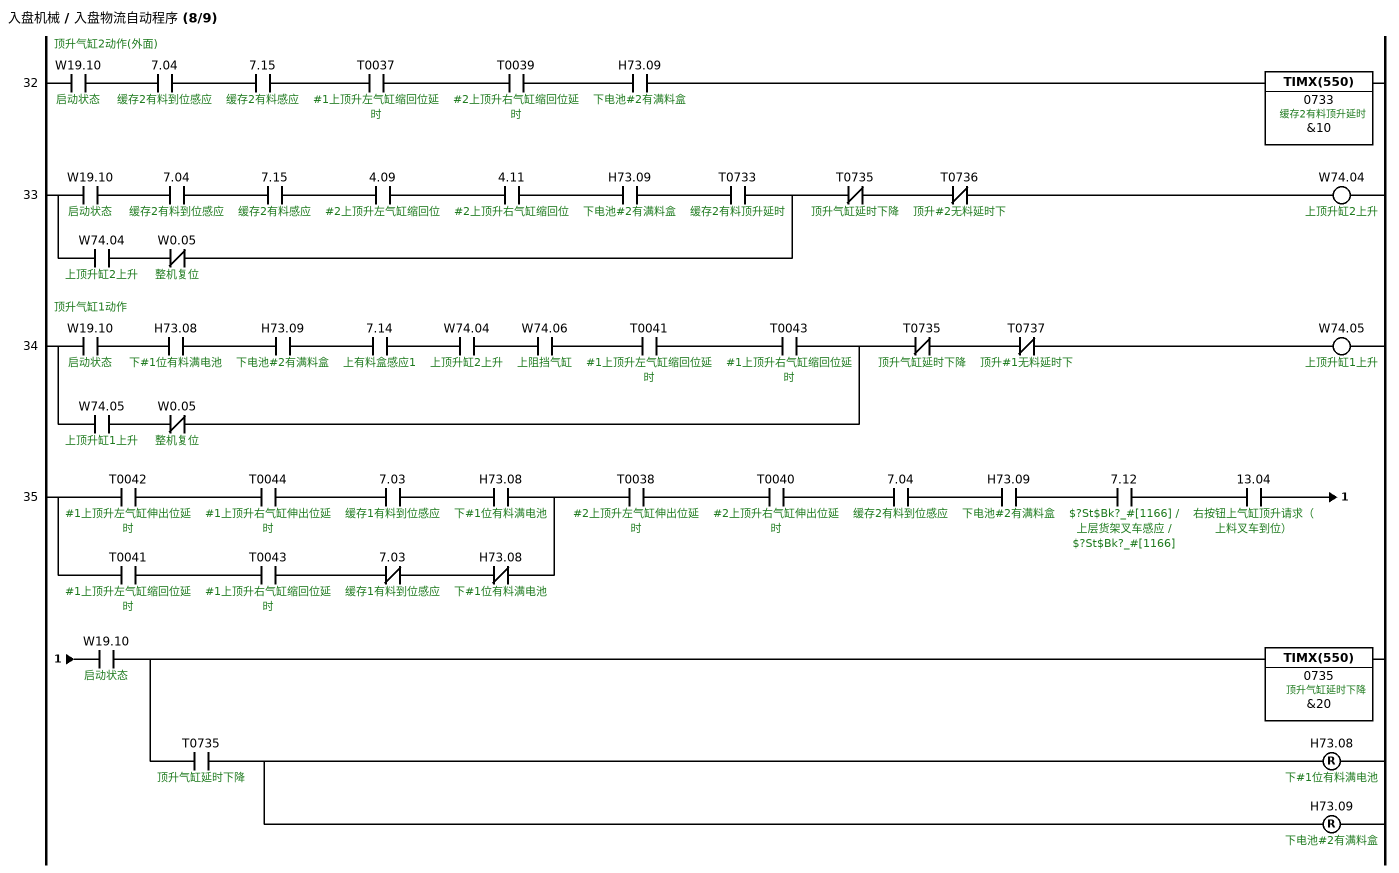
; [picture p240: 入盘机械 / 入盘物流自动程序, rungs 32-35]
; rung 32: 顶升气缸2动作(外面)
LD W19.10  ; 启动状态
AND 7.04  ; 缓存2有料到位感应
AND 7.15  ; 缓存2有料感应
AND T0037  ; #1上顶升左气缸缩回位延时
AND T0039  ; #2上顶升右气缸缩回位延时
AND H73.09  ; 下电池#2有满料盒
TIMX(550) 0733 &10  ; 缓存2有料顶升延时
; rung 33
LD W19.10  ; 启动状态
AND 7.04  ; 缓存2有料到位感应
AND 7.15  ; 缓存2有料感应
AND 4.09  ; #2上顶升左气缸缩回位
AND 4.11  ; #2上顶升右气缸缩回位
AND H73.09  ; 下电池#2有满料盒
AND T0733  ; 缓存2有料顶升延时
LD W74.04  ; 上顶升缸2上升
ANDNOT W0.05  ; 整机复位
ORLD
ANDNOT T0735  ; 顶升气缸延时下降
ANDNOT T0736  ; 顶升#2无料延时下
OUT W74.04  ; 上顶升缸2上升
; rung 34: 顶升气缸1动作
LD W19.10  ; 启动状态
AND H73.08  ; 下#1位有料满电池
AND H73.09  ; 下电池#2有满料盒
AND 7.14  ; 上有料盒感应1
AND W74.04  ; 上顶升缸2上升
AND W74.06  ; 上阻挡气缸
AND T0041  ; #1上顶升左气缸缩回位延时
AND T0043  ; #1上顶升右气缸缩回位延时
LD W74.05  ; 上顶升缸1上升
ANDNOT W0.05  ; 整机复位
ORLD
ANDNOT T0735  ; 顶升气缸延时下降
ANDNOT T0737  ; 顶升#1无料延时下
OUT W74.05  ; 上顶升缸1上升
; rung 35
LD T0042  ; #1上顶升左气缸伸出位延时
AND T0044  ; #1上顶升右气缸伸出位延时
AND 7.03  ; 缓存1有料到位感应
AND H73.08  ; 下#1位有料满电池
LD T0041  ; #1上顶升左气缸缩回位延时
AND T0043  ; #1上顶升右气缸缩回位延时
ANDNOT 7.03  ; 缓存1有料到位感应
ANDNOT H73.08  ; 下#1位有料满电池
ORLD
AND T0038  ; #2上顶升左气缸伸出位延时
AND T0040  ; #2上顶升右气缸伸出位延时
AND 7.04  ; 缓存2有料到位感应
AND H73.09  ; 下电池#2有满料盒
AND 7.12  ; $?St$Bk?_#[1166] / 上层货架叉车感应 / $?St$Bk?_#[1166]
AND 13.04  ; 右按钮上气缸顶升请求（上料叉车到位）
AND W19.10  ; 启动状态
TIMX(550) 0735 &20  ; 顶升气缸延时下降
AND T0735  ; 顶升气缸延时下降
RSET H73.08  ; 下#1位有料满电池
RSET H73.09  ; 下电池#2有满料盒

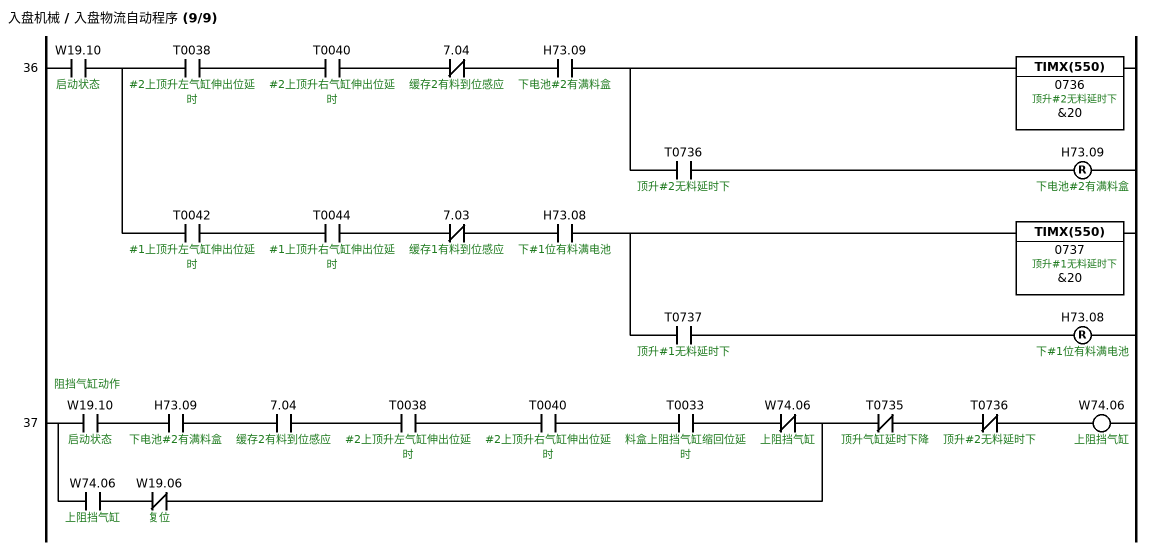
; rung 36
LD W19.10  ; 启动状态
OUT TR0
AND T0038  ; #2上顶升左气缸伸出位延时
AND T0040  ; #2上顶升右气缸伸出位延时
ANDNOT 7.04  ; 缓存2有料到位感应
AND H73.09  ; 下电池#2有满料盒
TIMX(550) 0736 &20  ; 顶升#2无料延时下
AND T0736  ; 顶升#2无料延时下
RSET H73.09  ; 下电池#2有满料盒
LD TR0
AND T0042  ; #1上顶升左气缸伸出位延时
AND T0044  ; #1上顶升右气缸伸出位延时
ANDNOT 7.03  ; 缓存1有料到位感应
AND H73.08  ; 下#1位有料满电池
TIMX(550) 0737 &20  ; 顶升#1无料延时下
AND T0737  ; 顶升#1无料延时下
RSET H73.08  ; 下#1位有料满电池
; rung 37: 阻挡气缸动作
LD W19.10  ; 启动状态
AND H73.09  ; 下电池#2有满料盒
AND 7.04  ; 缓存2有料到位感应
AND T0038  ; #2上顶升左气缸伸出位延时
AND T0040  ; #2上顶升右气缸伸出位延时
AND T0033  ; 料盒上阻挡气缸缩回位延时
ANDNOT W74.06  ; 上阻挡气缸
LD W74.06  ; 上阻挡气缸
ANDNOT W19.06  ; 复位
ORLD
ANDNOT T0735  ; 顶升气缸延时下降
ANDNOT T0736  ; 顶升#2无料延时下
OUT W74.06  ; 上阻挡气缸

### Section 伺服参数设定

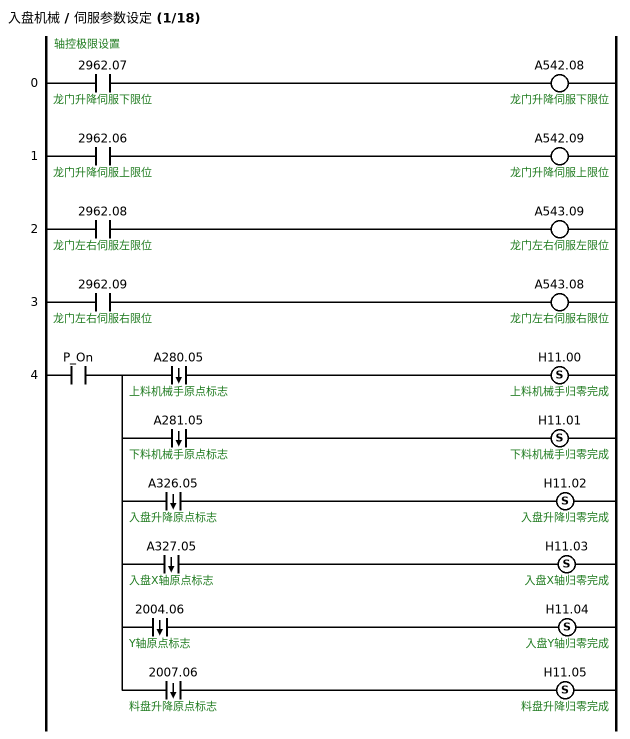
; rung 0: 轴控极限设置
LD 2962.07  ; 龙门升降伺服下限位
OUT A542.08  ; 龙门升降伺服下限位
; rung 1
LD 2962.06  ; 龙门升降伺服上限位
OUT A542.09  ; 龙门升降伺服上限位
; rung 2
LD 2962.08  ; 龙门左右伺服左限位
OUT A543.09  ; 龙门左右伺服左限位
; rung 3
LD 2962.09  ; 龙门左右伺服右限位
OUT A543.08  ; 龙门左右伺服右限位
; rung 4
LD P_On
OUT TR0
%AND A280.05  ; 上料机械手原点标志
SET H11.00  ; 上料机械手归零完成
LD TR0
%AND A281.05  ; 下料机械手原点标志
SET H11.01  ; 下料机械手归零完成
LD TR0
%AND A326.05  ; 入盘升降原点标志
SET H11.02  ; 入盘升降归零完成
LD TR0
%AND A327.05  ; 入盘X轴原点标志
SET H11.03  ; 入盘X轴归零完成
LD TR0
%AND 2004.06  ; Y轴原点标志
SET H11.04  ; 入盘Y轴归零完成
LD TR0
%AND 2007.06  ; 料盘升降原点标志
SET H11.05  ; 料盘升降归零完成

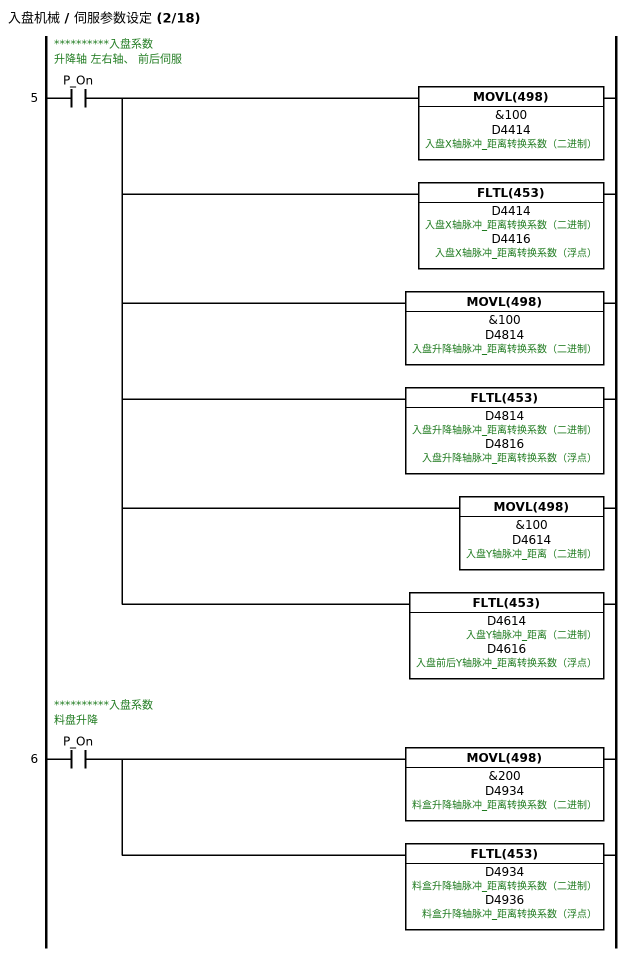
; rung 5: **********入盘系数 / 升降轴 左右轴、 前后伺服
LD P_On
MOVL(498) &100 D4414  ; 入盘X轴脉冲_距离转换系数（二进制）
FLTL(453) D4414 D4416  ; 入盘X轴脉冲_距离转换系数（二进制）, 入盘X轴脉冲_距离转换系数（浮点）
MOVL(498) &100 D4814  ; 入盘升降轴脉冲_距离转换系数（二进制）
FLTL(453) D4814 D4816  ; 入盘升降轴脉冲_距离转换系数（二进制）, 入盘升降轴脉冲_距离转换系数（浮点）
MOVL(498) &100 D4614  ; 入盘Y轴脉冲_距离（二进制）
FLTL(453) D4614 D4616  ; 入盘Y轴脉冲_距离（二进制）, 入盘前后Y轴脉冲_距离转换系数（浮点）
; rung 6: **********入盘系数 / 料盘升降
LD P_On
MOVL(498) &200 D4934  ; 料盒升降轴脉冲_距离转换系数（二进制）
FLTL(453) D4934 D4936  ; 料盒升降轴脉冲_距离转换系数（二进制）, 料盒升降轴脉冲_距离转换系数（浮点）

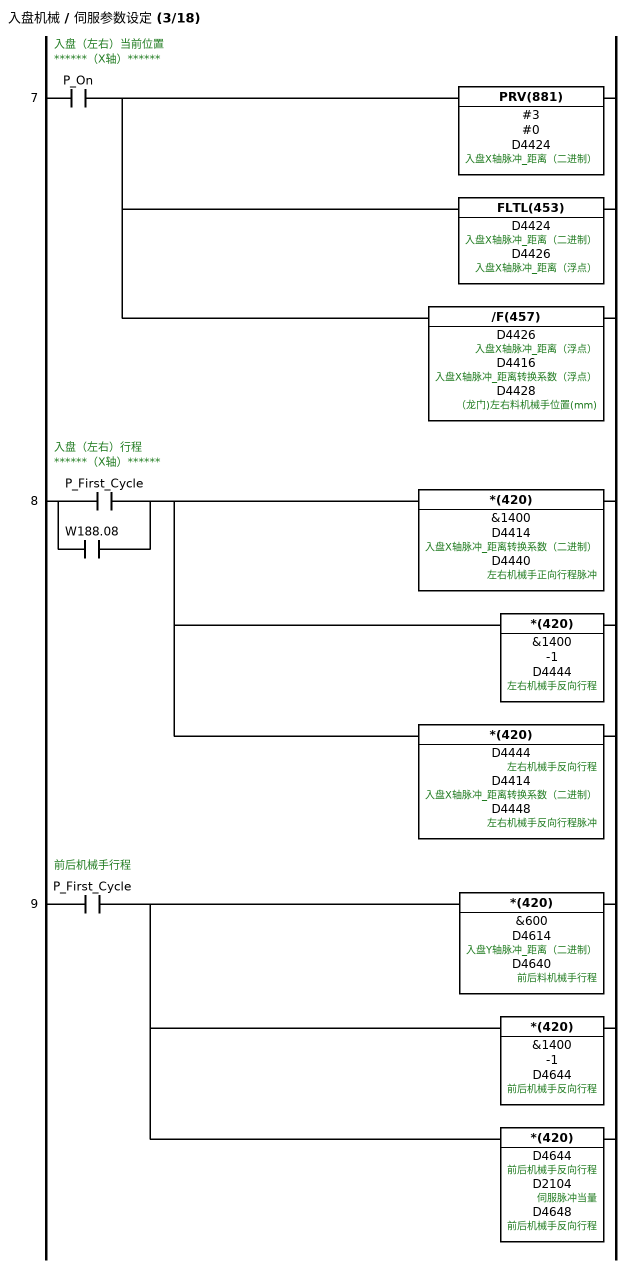
; rung 7: 入盘（左右）当前位置 / ******（X轴）******
LD P_On
PRV(881) #3 #0 D4424  ; 入盘X轴脉冲_距离（二进制）
FLTL(453) D4424 D4426  ; 入盘X轴脉冲_距离（二进制）, 入盘X轴脉冲_距离（浮点）
/F(457) D4426 D4416 D4428  ; 入盘X轴脉冲_距离（浮点）, 入盘X轴脉冲_距离转换系数（浮点）, （龙门)左右料机械手位置(mm)
; rung 8: 入盘（左右）行程 / ******（X轴）******
LD P_First_Cycle
OR W188.08
*(420) &1400 D4414 D4440  ; 入盘X轴脉冲_距离转换系数（二进制）, 左右机械手正向行程脉冲
*(420) &1400 -1 D4444  ; 左右机械手反向行程
*(420) D4444 D4414 D4448  ; 左右机械手反向行程, 入盘X轴脉冲_距离转换系数（二进制）, 左右机械手反向行程脉冲
; rung 9: 前后机械手行程
LD P_First_Cycle
*(420) &600 D4614 D4640  ; 入盘Y轴脉冲_距离（二进制）, 前后料机械手行程
*(420) &1400 -1 D4644  ; 前后机械手反向行程
*(420) D4644 D2104 D4648  ; 前后机械手反向行程, 伺服脉冲当量

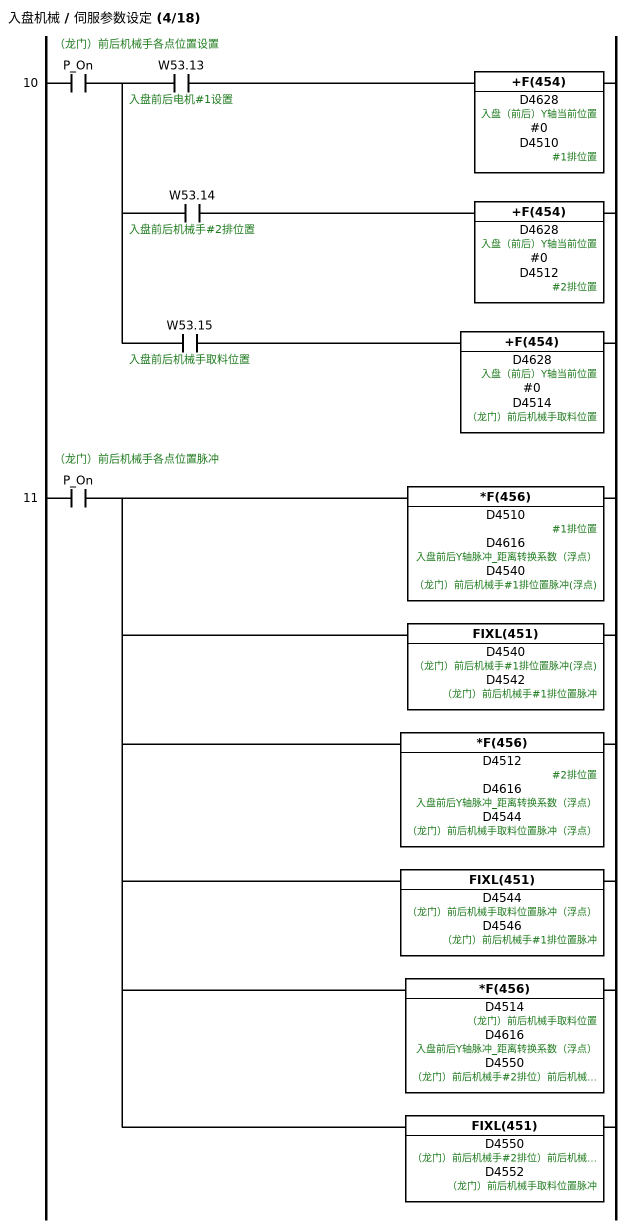
; rung 10: （龙门）前后机械手各点位置设置
LD P_On
OUT TR0
AND W53.13  ; 入盘前后电机#1设置
+F(454) D4628 #0 D4510  ; 入盘（前后）Y轴当前位置, #1排位置
LD TR0
AND W53.14  ; 入盘前后机械手#2排位置
+F(454) D4628 #0 D4512  ; 入盘（前后）Y轴当前位置, #2排位置
LD TR0
AND W53.15  ; 入盘前后机械手取料位置
+F(454) D4628 #0 D4514  ; 入盘（前后）Y轴当前位置, （龙门）前后机械手取料位置
; rung 11: （龙门）前后机械手各点位置脉冲
LD P_On
*F(456) D4510 D4616 D4540  ; #1排位置, 入盘前后Y轴脉冲_距离转换系数（浮点）, （龙门）前后机械手#1排位置脉冲(浮点)
FIXL(451) D4540 D4542  ; （龙门）前后机械手#1排位置脉冲(浮点), （龙门）前后机械手#1排位置脉冲
*F(456) D4512 D4616 D4544  ; #2排位置, 入盘前后Y轴脉冲_距离转换系数（浮点）, （龙门）前后机械手取料位置脉冲（浮点）
FIXL(451) D4544 D4546  ; （龙门）前后机械手取料位置脉冲（浮点）, （龙门）前后机械手#1排位置脉冲
*F(456) D4514 D4616 D4550  ; （龙门）前后机械手取料位置, 入盘前后Y轴脉冲_距离转换系数（浮点）, （龙门）前后机械手#2排位）前后机械手取料位(浮点)
FIXL(451) D4550 D4552  ; （龙门）前后机械手#2排位）前后机械手取料位(浮点), （龙门）前后机械手取料位置脉冲

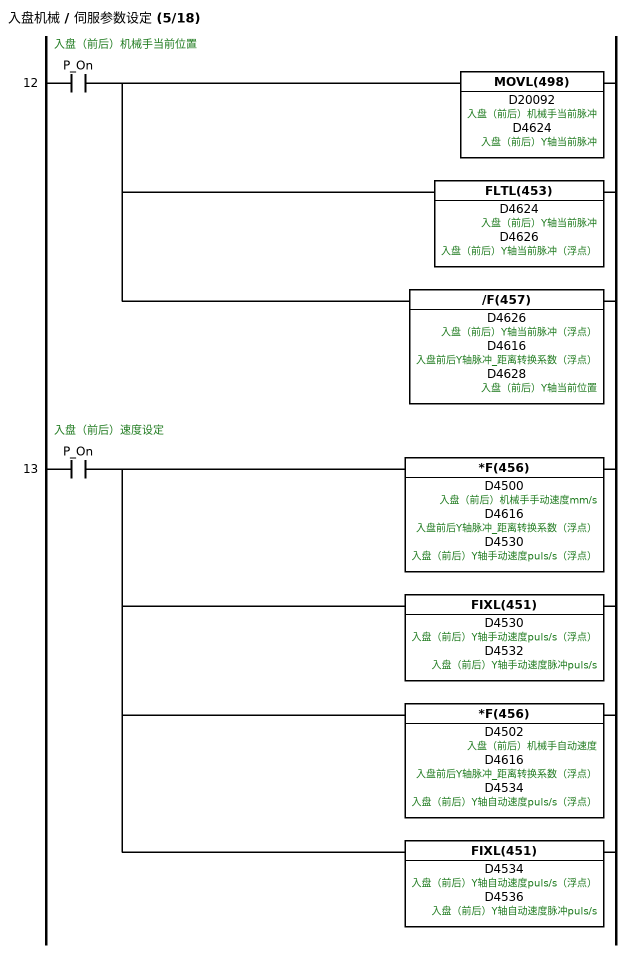
; rung 12: 入盘（前后）机械手当前位置
LD P_On
MOVL(498) D20092 D4624  ; 入盘（前后）机械手当前脉冲, 入盘（前后）Y轴当前脉冲
FLTL(453) D4624 D4626  ; 入盘（前后）Y轴当前脉冲, 入盘（前后）Y轴当前脉冲（浮点）
/F(457) D4626 D4616 D4628  ; 入盘（前后）Y轴当前脉冲（浮点）, 入盘前后Y轴脉冲_距离转换系数（浮点）, 入盘（前后）Y轴当前位置
; rung 13: 入盘（前后）速度设定
LD P_On
*F(456) D4500 D4616 D4530  ; 入盘（前后）机械手手动速度mm/s, 入盘前后Y轴脉冲_距离转换系数（浮点）, 入盘（前后）Y轴手动速度puls/s（浮点）
FIXL(451) D4530 D4532  ; 入盘（前后）Y轴手动速度puls/s（浮点）, 入盘（前后）Y轴手动速度脉冲puls/s
*F(456) D4502 D4616 D4534  ; 入盘（前后）机械手自动速度, 入盘前后Y轴脉冲_距离转换系数（浮点）, 入盘（前后）Y轴自动速度puls/s（浮点）
FIXL(451) D4534 D4536  ; 入盘（前后）Y轴自动速度puls/s（浮点）, 入盘（前后）Y轴自动速度脉冲puls/s

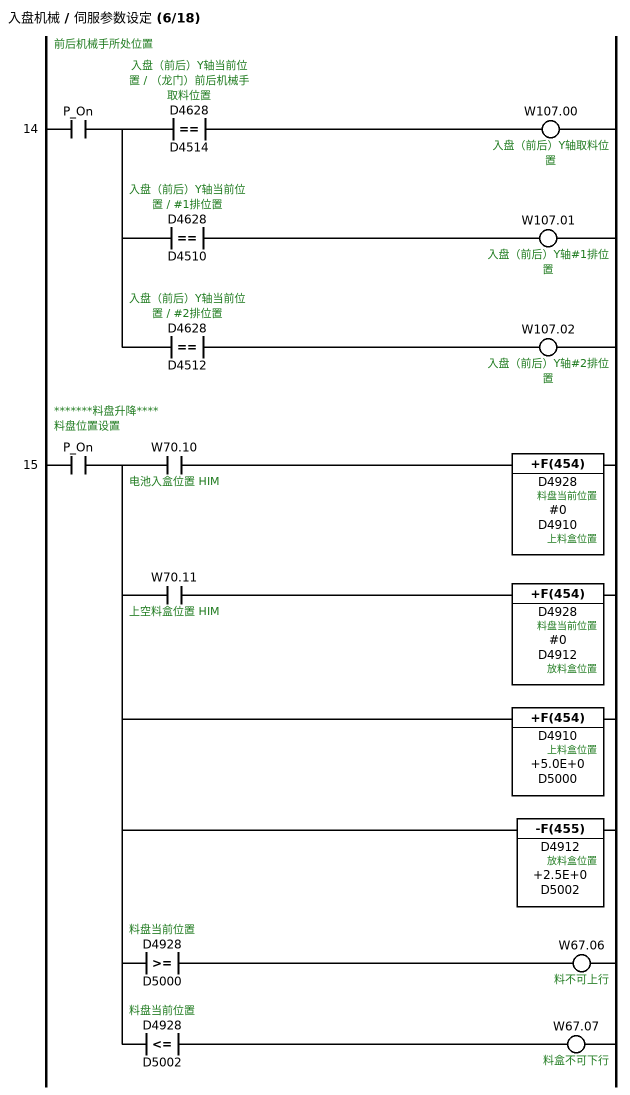
; rung 14: 前后机械手所处位置
LD P_On
OUT TR0
AND=SL(303) D4628 D4514  ; 入盘（前后）Y轴当前位置, （龙门）前后机械手取料位置
OUT W107.00  ; 入盘（前后）Y轴取料位置
LD TR0
AND=SL(303) D4628 D4510  ; 入盘（前后）Y轴当前位置, #1排位置
OUT W107.01  ; 入盘（前后）Y轴#1排位置
LD TR0
AND=SL(303) D4628 D4512  ; 入盘（前后）Y轴当前位置, #2排位置
OUT W107.02  ; 入盘（前后）Y轴#2排位置
; rung 15: *******料盘升降**** / 料盘位置设置
LD P_On
OUT TR0
AND W70.10  ; 电池入盒位置 HIM
+F(454) D4928 #0 D4910  ; 料盘当前位置, 上料盒位置
LD TR0
AND W70.11  ; 上空料盒位置 HIM
+F(454) D4928 #0 D4912  ; 料盘当前位置, 放料盒位置
LD TR0
+F(454) D4910 +5.0E+0 D5000  ; 上料盒位置
-F(455) D4912 +2.5E+0 D5002  ; 放料盒位置
AND>=F(334) D4928 D5000  ; 料盘当前位置
OUT W67.06  ; 料不可上行
LD TR0
AND<=F(332) D4928 D5002  ; 料盘当前位置
OUT W67.07  ; 料盒不可下行

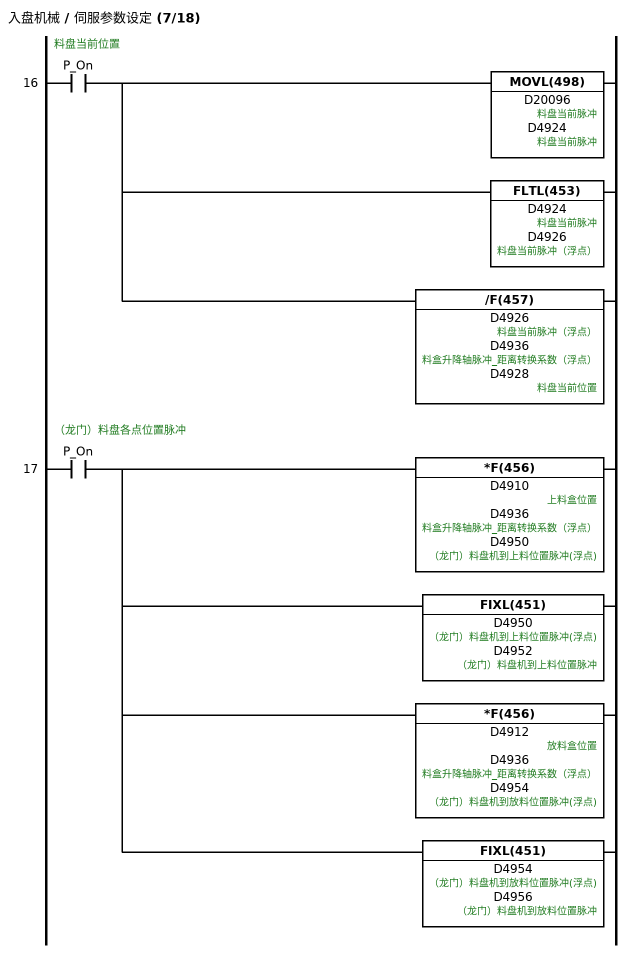
; rung 16: 料盘当前位置
LD P_On
MOVL(498) D20096 D4924  ; 料盘当前脉冲
FLTL(453) D4924 D4926  ; 料盘当前脉冲, 料盘当前脉冲（浮点）
/F(457) D4926 D4936 D4928  ; 料盘当前脉冲（浮点）, 料盒升降轴脉冲_距离转换系数（浮点）, 料盘当前位置
; rung 17: （龙门）料盘各点位置脉冲
LD P_On
*F(456) D4910 D4936 D4950  ; 上料盒位置, 料盒升降轴脉冲_距离转换系数（浮点）, （龙门）料盘机到上料位置脉冲(浮点)
FIXL(451) D4950 D4952  ; （龙门）料盘机到上料位置脉冲(浮点), （龙门）料盘机到上料位置脉冲
*F(456) D4912 D4936 D4954  ; 放料盒位置, 料盒升降轴脉冲_距离转换系数（浮点）, （龙门）料盘机到放料位置脉冲(浮点)
FIXL(451) D4954 D4956  ; （龙门）料盘机到放料位置脉冲(浮点), （龙门）料盘机到放料位置脉冲

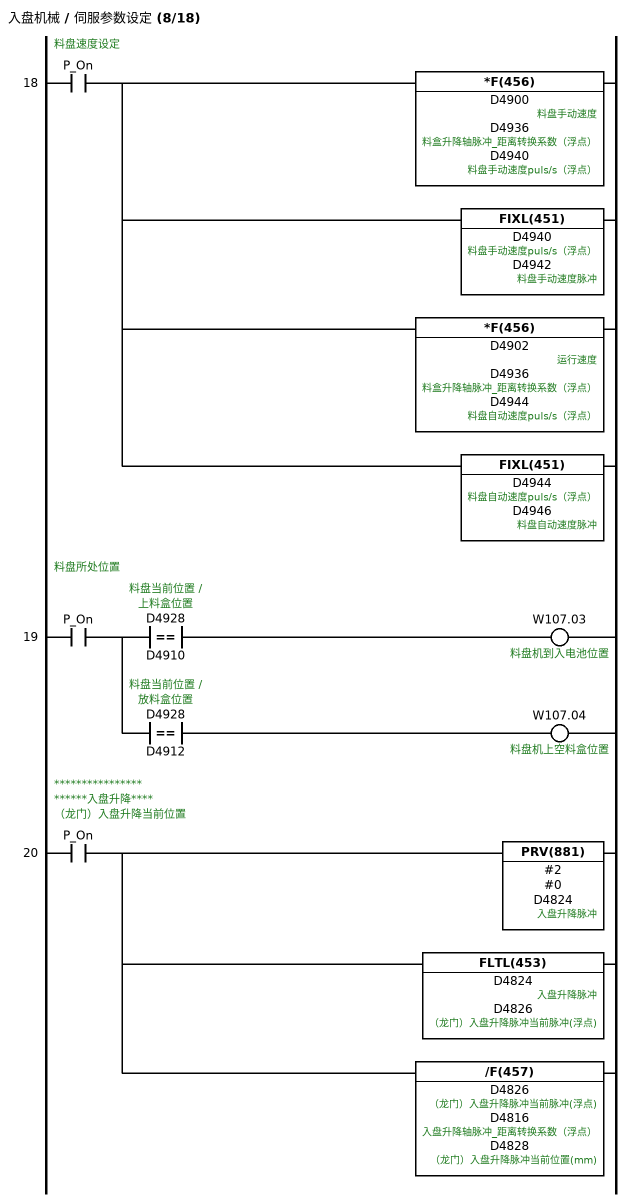
; rung 18: 料盘速度设定
LD P_On
*F(456) D4900 D4936 D4940  ; 料盘手动速度, 料盒升降轴脉冲_距离转换系数（浮点）, 料盘手动速度puls/s（浮点）
FIXL(451) D4940 D4942  ; 料盘手动速度puls/s（浮点）, 料盘手动速度脉冲
*F(456) D4902 D4936 D4944  ; 运行速度, 料盒升降轴脉冲_距离转换系数（浮点）, 料盘自动速度puls/s（浮点）
FIXL(451) D4944 D4946  ; 料盘自动速度puls/s（浮点）, 料盘自动速度脉冲
; rung 19: 料盘所处位置
LD P_On
OUT TR0
AND=SL(303) D4928 D4910  ; 料盘当前位置, 上料盒位置
OUT W107.03  ; 料盘机到入电池位置
LD TR0
AND=SL(303) D4928 D4912  ; 料盘当前位置, 放料盒位置
OUT W107.04  ; 料盘机上空料盒位置
; rung 20: **************** / ******入盘升降**** / （龙门）入盘升降当前位置
LD P_On
PRV(881) #2 #0 D4824  ; 入盘升降脉冲
FLTL(453) D4824 D4826  ; 入盘升降脉冲, （龙门）入盘升降脉冲当前脉冲(浮点)
/F(457) D4826 D4816 D4828  ; （龙门）入盘升降脉冲当前脉冲(浮点), 入盘升降轴脉冲_距离转换系数（浮点）, （龙门）入盘升降脉冲当前位置(mm)

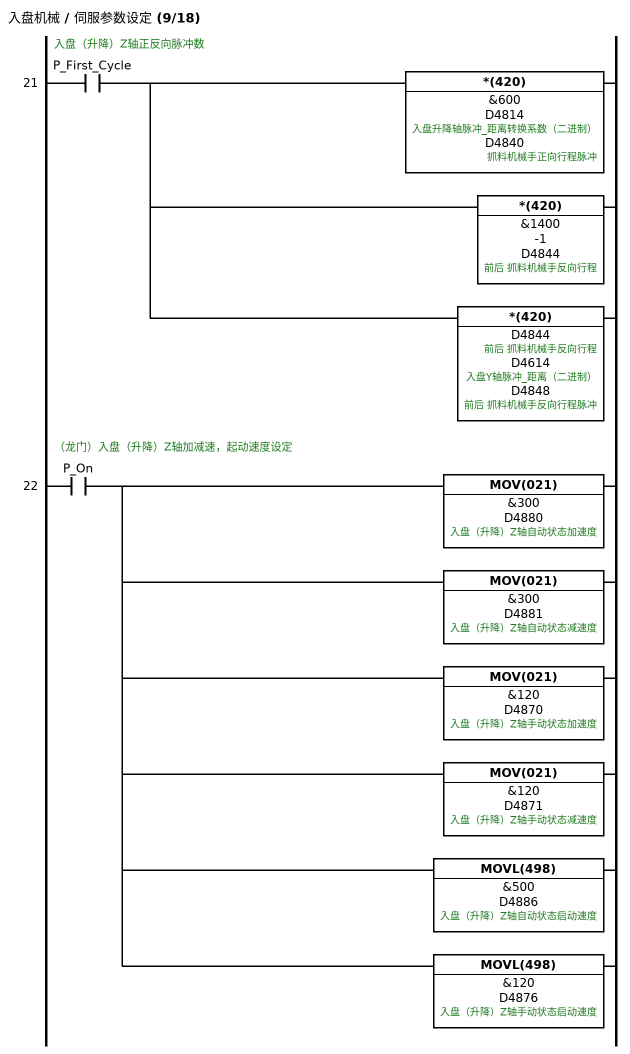
; rung 21: 入盘（升降）Z轴正反向脉冲数
LD P_First_Cycle
*(420) &600 D4814 D4840  ; 入盘升降轴脉冲_距离转换系数（二进制）, 抓料机械手正向行程脉冲
*(420) &1400 -1 D4844  ; 前后 抓料机械手反向行程
*(420) D4844 D4614 D4848  ; 前后 抓料机械手反向行程, 入盘Y轴脉冲_距离（二进制）, 前后 抓料机械手反向行程脉冲
; rung 22: （龙门）入盘（升降）Z轴加减速，起动速度设定
LD P_On
MOV(021) &300 D4880  ; 入盘（升降）Z轴自动状态加速度
MOV(021) &300 D4881  ; 入盘（升降）Z轴自动状态减速度
MOV(021) &120 D4870  ; 入盘（升降）Z轴手动状态加速度
MOV(021) &120 D4871  ; 入盘（升降）Z轴手动状态减速度
MOVL(498) &500 D4886  ; 入盘（升降）Z轴自动状态启动速度
MOVL(498) &120 D4876  ; 入盘（升降）Z轴手动状态启动速度

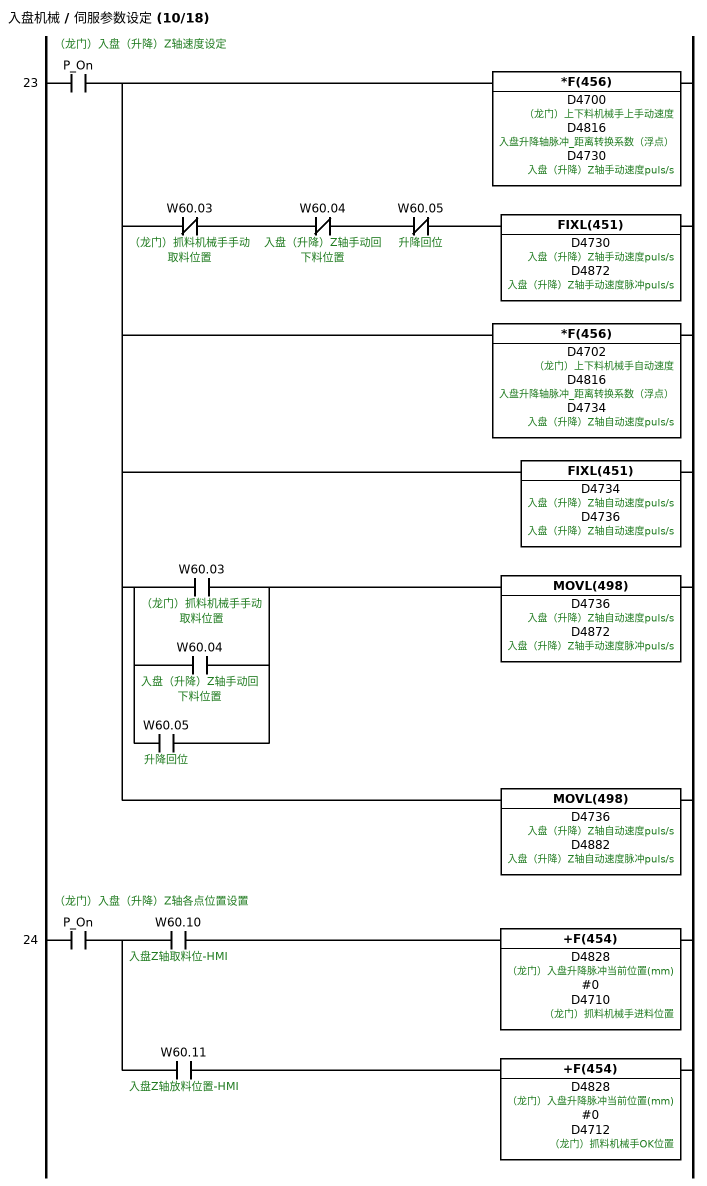
; rung 23: （龙门）入盘（升降）Z轴速度设定
LD P_On
OUT TR0
*F(456) D4700 D4816 D4730  ; （龙门）上下料机械手上手动速度, 入盘升降轴脉冲_距离转换系数（浮点）, 入盘（升降）Z轴手动速度puls/s
ANDNOT W60.03  ; （龙门）抓料机械手手动取料位置
ANDNOT W60.04  ; 入盘（升降）Z轴手动回下料位置
ANDNOT W60.05  ; 升降回位
FIXL(451) D4730 D4872  ; 入盘（升降）Z轴手动速度puls/s, 入盘（升降）Z轴手动速度脉冲puls/s
LD TR0
*F(456) D4702 D4816 D4734  ; （龙门）上下料机械手自动速度, 入盘升降轴脉冲_距离转换系数（浮点）, 入盘（升降）Z轴自动速度puls/s
FIXL(451) D4734 D4736  ; 入盘（升降）Z轴自动速度puls/s
LD W60.03  ; （龙门）抓料机械手手动取料位置
OR W60.04  ; 入盘（升降）Z轴手动回下料位置
OR W60.05  ; 升降回位
ANDLD
MOVL(498) D4736 D4872  ; 入盘（升降）Z轴自动速度puls/s, 入盘（升降）Z轴手动速度脉冲puls/s
LD TR0
MOVL(498) D4736 D4882  ; 入盘（升降）Z轴自动速度puls/s, 入盘（升降）Z轴自动速度脉冲puls/s
; rung 24: （龙门）入盘（升降）Z轴各点位置设置
LD P_On
OUT TR0
AND W60.10  ; 入盘Z轴取料位-HMI
+F(454) D4828 #0 D4710  ; （龙门）入盘升降脉冲当前位置(mm), （龙门）抓料机械手进料位置
LD TR0
AND W60.11  ; 入盘Z轴放料位置-HMI
+F(454) D4828 #0 D4712  ; （龙门）入盘升降脉冲当前位置(mm), （龙门）抓料机械手OK位置

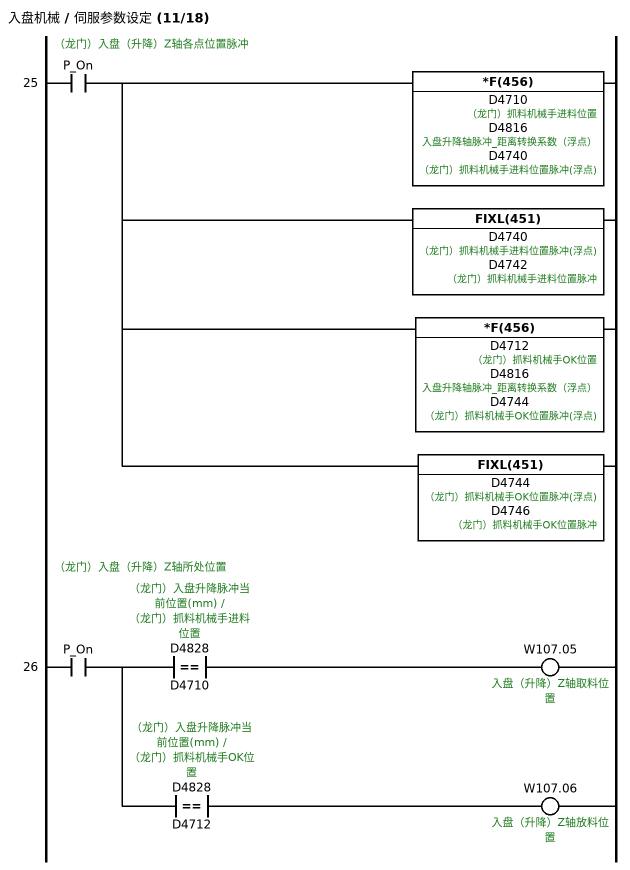
; rung 25: （龙门）入盘（升降）Z轴各点位置脉冲
LD P_On
*F(456) D4710 D4816 D4740  ; （龙门）抓料机械手进料位置, 入盘升降轴脉冲_距离转换系数（浮点）, （龙门）抓料机械手进料位置脉冲(浮点)
FIXL(451) D4740 D4742  ; （龙门）抓料机械手进料位置脉冲(浮点), （龙门）抓料机械手进料位置脉冲
*F(456) D4712 D4816 D4744  ; （龙门）抓料机械手OK位置, 入盘升降轴脉冲_距离转换系数（浮点）, （龙门）抓料机械手OK位置脉冲(浮点)
FIXL(451) D4744 D4746  ; （龙门）抓料机械手OK位置脉冲(浮点), （龙门）抓料机械手OK位置脉冲
; rung 26: （龙门）入盘（升降）Z轴所处位置
LD P_On
OUT TR0
AND=SL(303) D4828 D4710  ; （龙门）入盘升降脉冲当前位置(mm), （龙门）抓料机械手进料位置
OUT W107.05  ; 入盘（升降）Z轴取料位置
LD TR0
AND=SL(303) D4828 D4712  ; （龙门）入盘升降脉冲当前位置(mm), （龙门）抓料机械手OK位置
OUT W107.06  ; 入盘（升降）Z轴放料位置

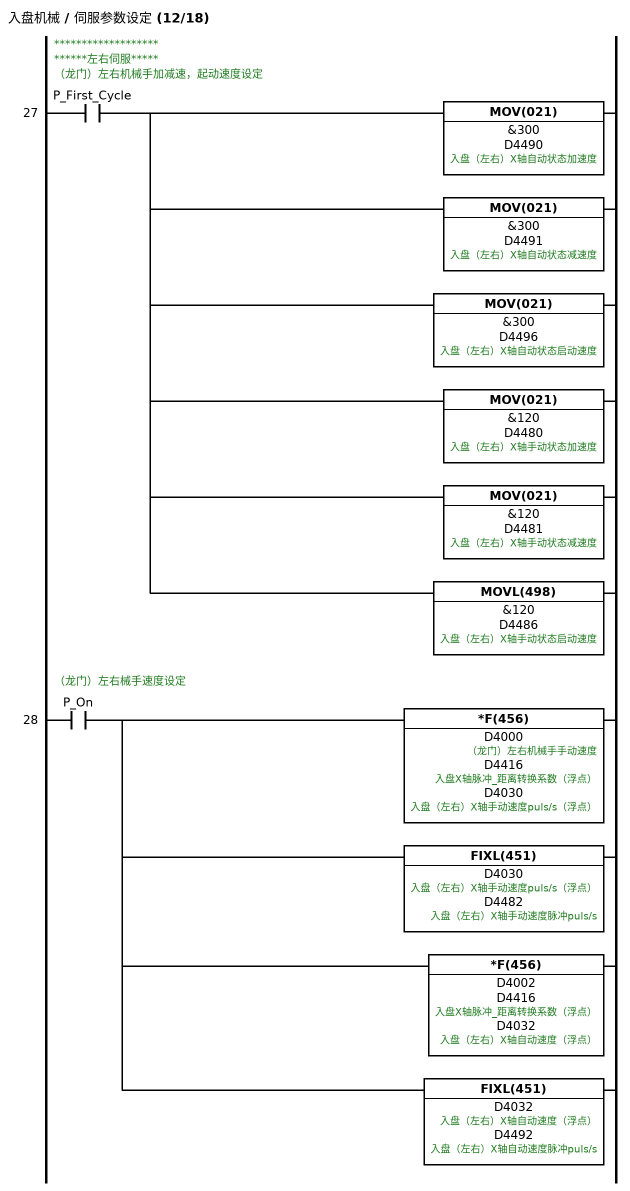
; rung 27: ******************* / ******左右伺服***** / （龙门）左右机械手加减速，起动速度设定
LD P_First_Cycle
MOV(021) &300 D4490  ; 入盘（左右）X轴自动状态加速度
MOV(021) &300 D4491  ; 入盘（左右）X轴自动状态减速度
MOV(021) &300 D4496  ; 入盘（左右）X轴自动状态启动速度
MOV(021) &120 D4480  ; 入盘（左右）X轴手动状态加速度
MOV(021) &120 D4481  ; 入盘（左右）X轴手动状态减速度
MOVL(498) &120 D4486  ; 入盘（左右）X轴手动状态启动速度
; rung 28: （龙门）左右械手速度设定
LD P_On
*F(456) D4000 D4416 D4030  ; （龙门）左右机械手手动速度, 入盘X轴脉冲_距离转换系数（浮点）, 入盘（左右）X轴手动速度puls/s（浮点）
FIXL(451) D4030 D4482  ; 入盘（左右）X轴手动速度puls/s（浮点）, 入盘（左右）X轴手动速度脉冲puls/s
*F(456) D4002 D4416 D4032  ; 入盘X轴脉冲_距离转换系数（浮点）, 入盘（左右）X轴自动速度（浮点）
FIXL(451) D4032 D4492  ; 入盘（左右）X轴自动速度（浮点）, 入盘（左右）X轴自动速度脉冲puls/s

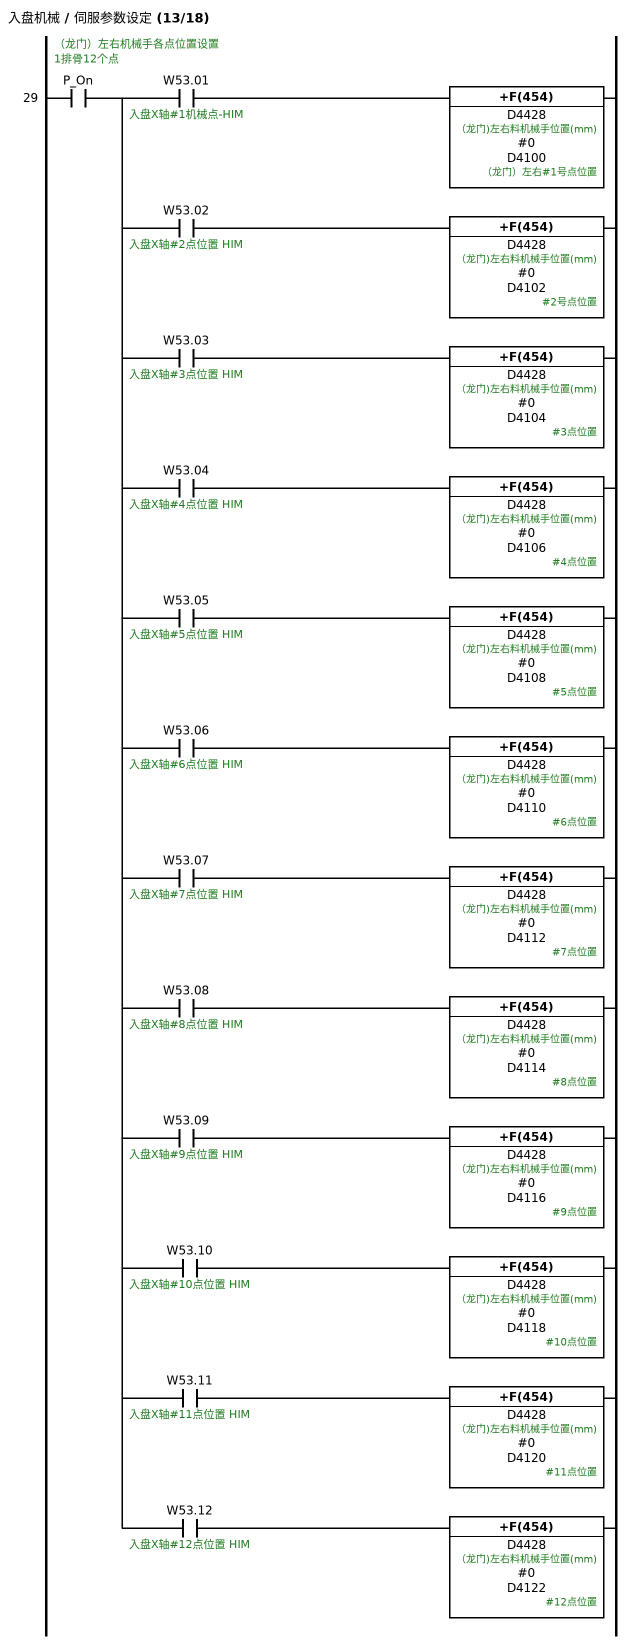
; rung 29: （龙门）左右机械手各点位置设置 / 1排骨12个点
LD P_On
OUT TR0
AND W53.01  ; 入盘X轴#1机械点-HIM
+F(454) D4428 #0 D4100  ; （龙门)左右料机械手位置(mm), （龙门）左右#1号点位置
LD TR0
AND W53.02  ; 入盘X轴#2点位置 HIM
+F(454) D4428 #0 D4102  ; （龙门)左右料机械手位置(mm), #2号点位置
LD TR0
AND W53.03  ; 入盘X轴#3点位置 HIM
+F(454) D4428 #0 D4104  ; （龙门)左右料机械手位置(mm), #3点位置
LD TR0
AND W53.04  ; 入盘X轴#4点位置 HIM
+F(454) D4428 #0 D4106  ; （龙门)左右料机械手位置(mm), #4点位置
LD TR0
AND W53.05  ; 入盘X轴#5点位置 HIM
+F(454) D4428 #0 D4108  ; （龙门)左右料机械手位置(mm), #5点位置
LD TR0
AND W53.06  ; 入盘X轴#6点位置 HIM
+F(454) D4428 #0 D4110  ; （龙门)左右料机械手位置(mm), #6点位置
LD TR0
AND W53.07  ; 入盘X轴#7点位置 HIM
+F(454) D4428 #0 D4112  ; （龙门)左右料机械手位置(mm), #7点位置
LD TR0
AND W53.08  ; 入盘X轴#8点位置 HIM
+F(454) D4428 #0 D4114  ; （龙门)左右料机械手位置(mm), #8点位置
LD TR0
AND W53.09  ; 入盘X轴#9点位置 HIM
+F(454) D4428 #0 D4116  ; （龙门)左右料机械手位置(mm), #9点位置
LD TR0
AND W53.10  ; 入盘X轴#10点位置 HIM
+F(454) D4428 #0 D4118  ; （龙门)左右料机械手位置(mm), #10点位置
LD TR0
AND W53.11  ; 入盘X轴#11点位置 HIM
+F(454) D4428 #0 D4120  ; （龙门)左右料机械手位置(mm), #11点位置
LD TR0
AND W53.12  ; 入盘X轴#12点位置 HIM
+F(454) D4428 #0 D4122  ; （龙门)左右料机械手位置(mm), #12点位置

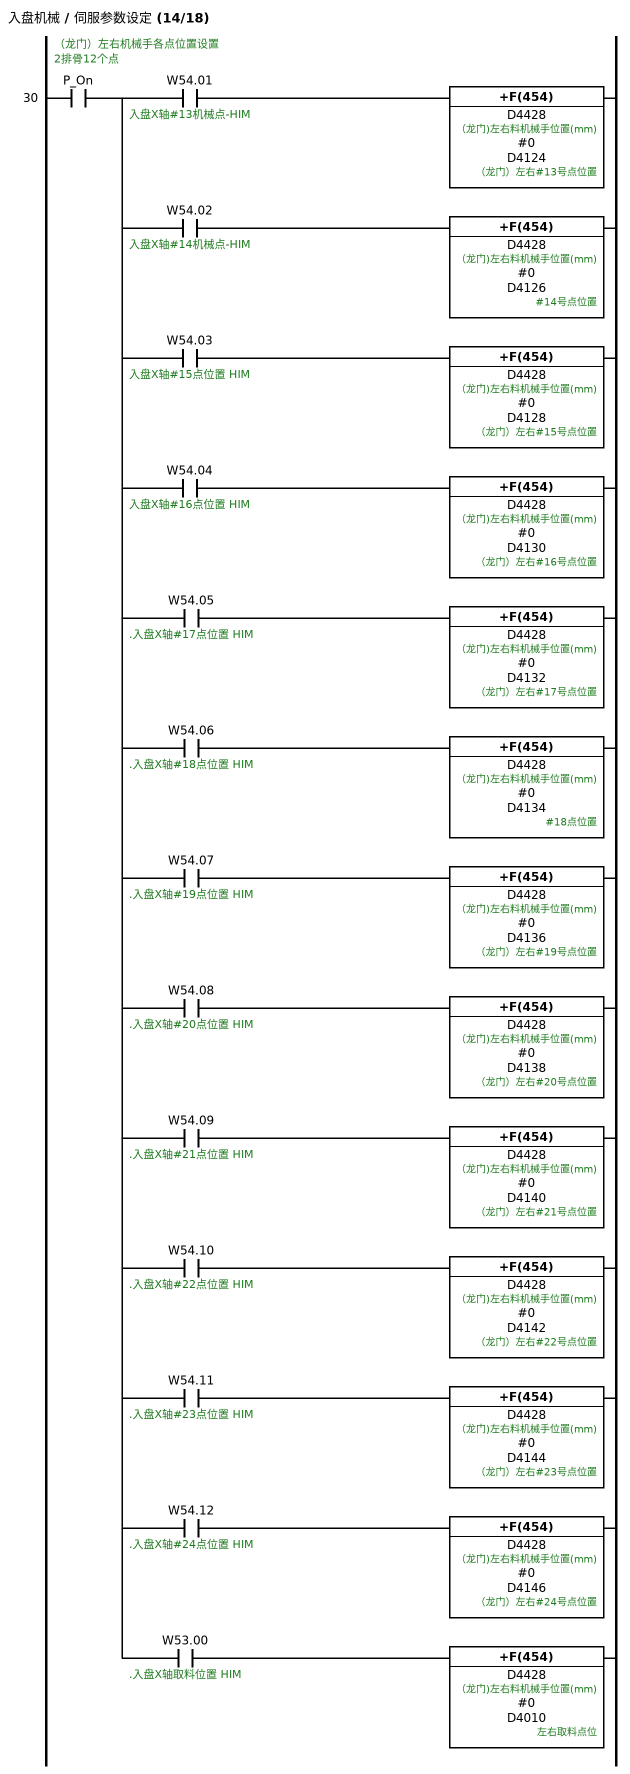
; rung 30: （龙门）左右机械手各点位置设置 / 2排骨12个点
LD P_On
OUT TR0
AND W54.01  ; 入盘X轴#13机械点-HIM
+F(454) D4428 #0 D4124  ; （龙门)左右料机械手位置(mm), （龙门）左右#13号点位置
LD TR0
AND W54.02  ; 入盘X轴#14机械点-HIM
+F(454) D4428 #0 D4126  ; （龙门)左右料机械手位置(mm), #14号点位置
LD TR0
AND W54.03  ; 入盘X轴#15点位置 HIM
+F(454) D4428 #0 D4128  ; （龙门)左右料机械手位置(mm), （龙门）左右#15号点位置
LD TR0
AND W54.04  ; 入盘X轴#16点位置 HIM
+F(454) D4428 #0 D4130  ; （龙门)左右料机械手位置(mm), （龙门）左右#16号点位置
LD TR0
AND W54.05  ; .入盘X轴#17点位置 HIM
+F(454) D4428 #0 D4132  ; （龙门)左右料机械手位置(mm), （龙门）左右#17号点位置
LD TR0
AND W54.06  ; .入盘X轴#18点位置 HIM
+F(454) D4428 #0 D4134  ; （龙门)左右料机械手位置(mm), #18点位置
LD TR0
AND W54.07  ; .入盘X轴#19点位置 HIM
+F(454) D4428 #0 D4136  ; （龙门)左右料机械手位置(mm), （龙门）左右#19号点位置
LD TR0
AND W54.08  ; .入盘X轴#20点位置 HIM
+F(454) D4428 #0 D4138  ; （龙门)左右料机械手位置(mm), （龙门）左右#20号点位置
LD TR0
AND W54.09  ; .入盘X轴#21点位置 HIM
+F(454) D4428 #0 D4140  ; （龙门)左右料机械手位置(mm), （龙门）左右#21号点位置
LD TR0
AND W54.10  ; .入盘X轴#22点位置 HIM
+F(454) D4428 #0 D4142  ; （龙门)左右料机械手位置(mm), （龙门）左右#22号点位置
LD TR0
AND W54.11  ; .入盘X轴#23点位置 HIM
+F(454) D4428 #0 D4144  ; （龙门)左右料机械手位置(mm), （龙门）左右#23号点位置
LD TR0
AND W54.12  ; .入盘X轴#24点位置 HIM
+F(454) D4428 #0 D4146  ; （龙门)左右料机械手位置(mm), （龙门）左右#24号点位置
LD TR0
AND W53.00  ; .入盘X轴取料位置 HIM
+F(454) D4428 #0 D4010  ; （龙门)左右料机械手位置(mm), 左右取料点位

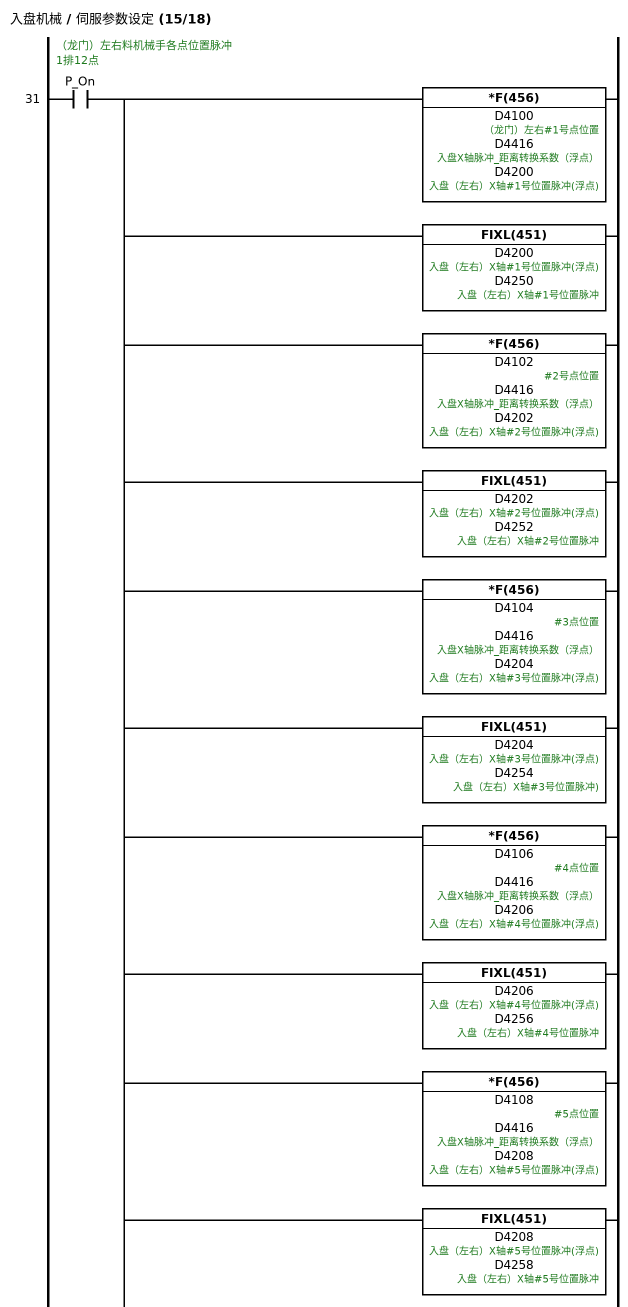

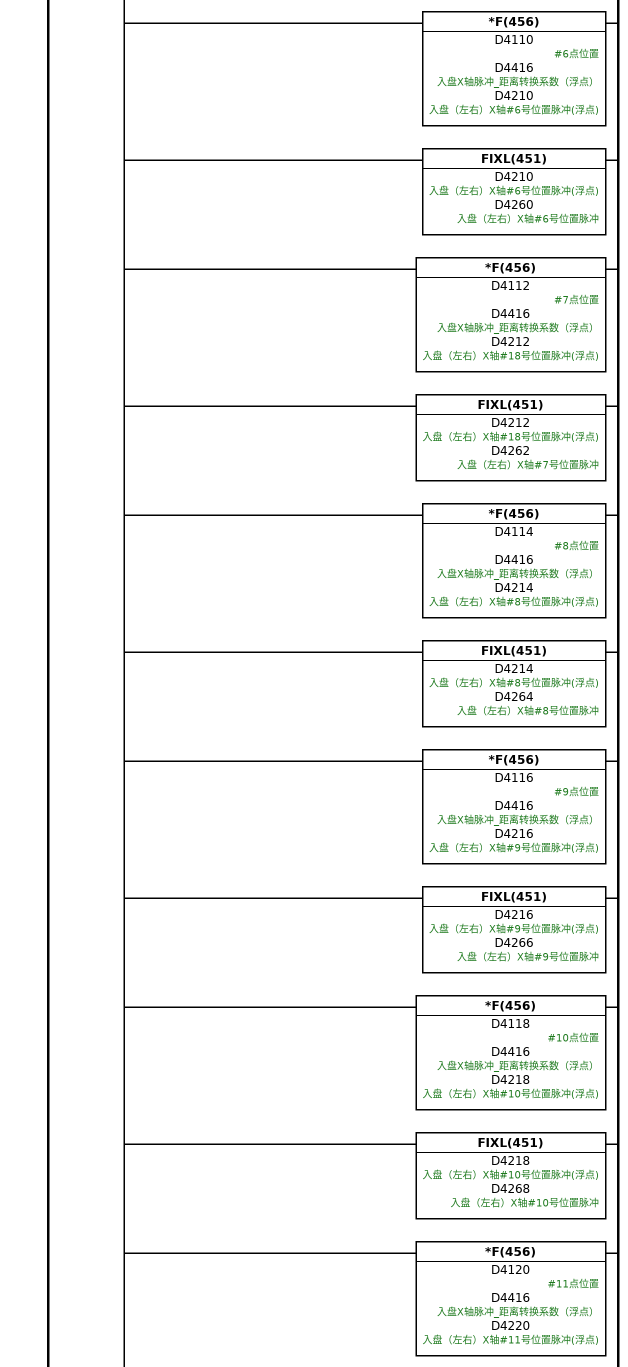

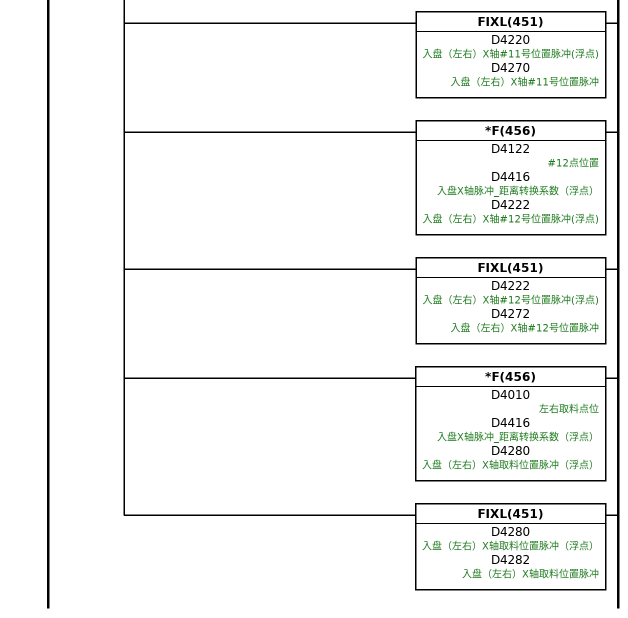
; rung 31: （龙门）左右料机械手各点位置脉冲 / 1排12点
LD P_On
*F(456) D4100 D4416 D4200  ; （龙门）左右#1号点位置, 入盘X轴脉冲_距离转换系数（浮点）, 入盘（左右）X轴#1号位置脉冲(浮点)
FIXL(451) D4200 D4250  ; 入盘（左右）X轴#1号位置脉冲(浮点), 入盘（左右）X轴#1号位置脉冲
*F(456) D4102 D4416 D4202  ; #2号点位置, 入盘X轴脉冲_距离转换系数（浮点）, 入盘（左右）X轴#2号位置脉冲(浮点)
FIXL(451) D4202 D4252  ; 入盘（左右）X轴#2号位置脉冲(浮点), 入盘（左右）X轴#2号位置脉冲
*F(456) D4104 D4416 D4204  ; #3点位置, 入盘X轴脉冲_距离转换系数（浮点）, 入盘（左右）X轴#3号位置脉冲(浮点)
FIXL(451) D4204 D4254  ; 入盘（左右）X轴#3号位置脉冲(浮点), 入盘（左右）X轴#3号位置脉冲)
*F(456) D4106 D4416 D4206  ; #4点位置, 入盘X轴脉冲_距离转换系数（浮点）, 入盘（左右）X轴#4号位置脉冲(浮点)
FIXL(451) D4206 D4256  ; 入盘（左右）X轴#4号位置脉冲(浮点), 入盘（左右）X轴#4号位置脉冲
*F(456) D4108 D4416 D4208  ; #5点位置, 入盘X轴脉冲_距离转换系数（浮点）, 入盘（左右）X轴#5号位置脉冲(浮点)
FIXL(451) D4208 D4258  ; 入盘（左右）X轴#5号位置脉冲(浮点), 入盘（左右）X轴#5号位置脉冲
*F(456) D4110 D4416 D4210  ; #6点位置, 入盘X轴脉冲_距离转换系数（浮点）, 入盘（左右）X轴#6号位置脉冲(浮点)
FIXL(451) D4210 D4260  ; 入盘（左右）X轴#6号位置脉冲(浮点), 入盘（左右）X轴#6号位置脉冲
*F(456) D4112 D4416 D4212  ; #7点位置, 入盘X轴脉冲_距离转换系数（浮点）, 入盘（左右）X轴#18号位置脉冲(浮点)
FIXL(451) D4212 D4262  ; 入盘（左右）X轴#18号位置脉冲(浮点), 入盘（左右）X轴#7号位置脉冲
*F(456) D4114 D4416 D4214  ; #8点位置, 入盘X轴脉冲_距离转换系数（浮点）, 入盘（左右）X轴#8号位置脉冲(浮点)
FIXL(451) D4214 D4264  ; 入盘（左右）X轴#8号位置脉冲(浮点), 入盘（左右）X轴#8号位置脉冲
*F(456) D4116 D4416 D4216  ; #9点位置, 入盘X轴脉冲_距离转换系数（浮点）, 入盘（左右）X轴#9号位置脉冲(浮点)
FIXL(451) D4216 D4266  ; 入盘（左右）X轴#9号位置脉冲(浮点), 入盘（左右）X轴#9号位置脉冲
*F(456) D4118 D4416 D4218  ; #10点位置, 入盘X轴脉冲_距离转换系数（浮点）, 入盘（左右）X轴#10号位置脉冲(浮点)
FIXL(451) D4218 D4268  ; 入盘（左右）X轴#10号位置脉冲(浮点), 入盘（左右）X轴#10号位置脉冲
*F(456) D4120 D4416 D4220  ; #11点位置, 入盘X轴脉冲_距离转换系数（浮点）, 入盘（左右）X轴#11号位置脉冲(浮点)
FIXL(451) D4220 D4270  ; 入盘（左右）X轴#11号位置脉冲(浮点), 入盘（左右）X轴#11号位置脉冲
*F(456) D4122 D4416 D4222  ; #12点位置, 入盘X轴脉冲_距离转换系数（浮点）, 入盘（左右）X轴#12号位置脉冲(浮点)
FIXL(451) D4222 D4272  ; 入盘（左右）X轴#12号位置脉冲(浮点), 入盘（左右）X轴#12号位置脉冲
*F(456) D4010 D4416 D4280  ; 左右取料点位, 入盘X轴脉冲_距离转换系数（浮点）, 入盘（左右）X轴取料位置脉冲（浮点）
FIXL(451) D4280 D4282  ; 入盘（左右）X轴取料位置脉冲（浮点）, 入盘（左右）X轴取料位置脉冲

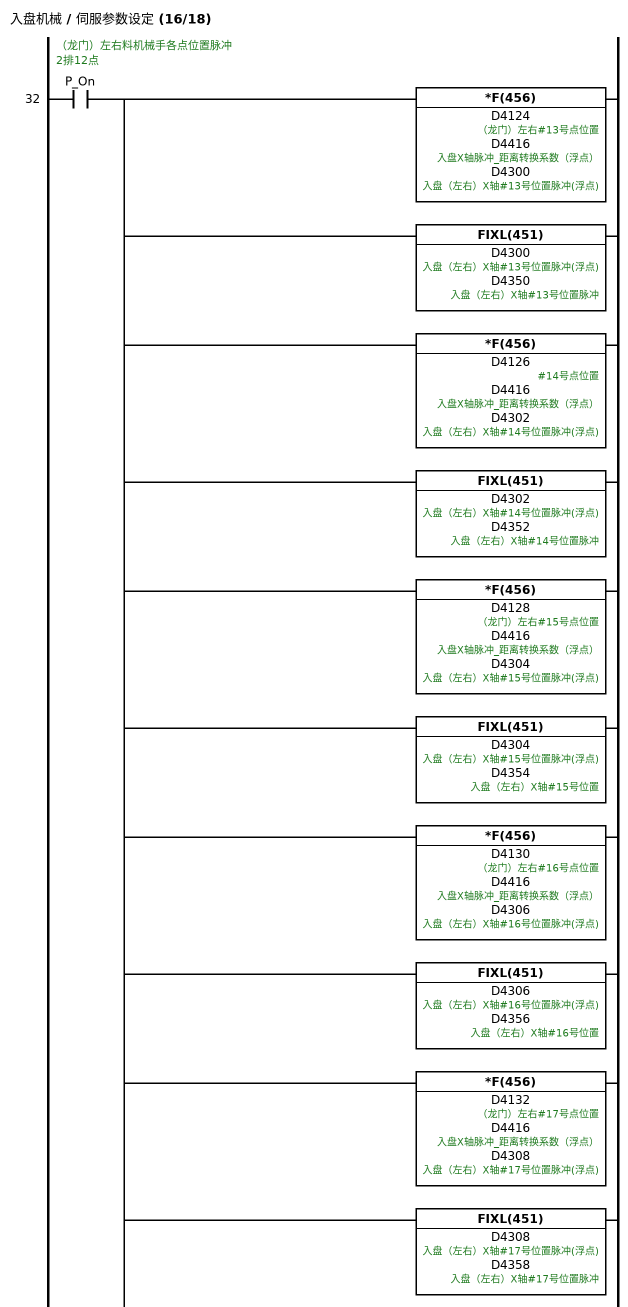

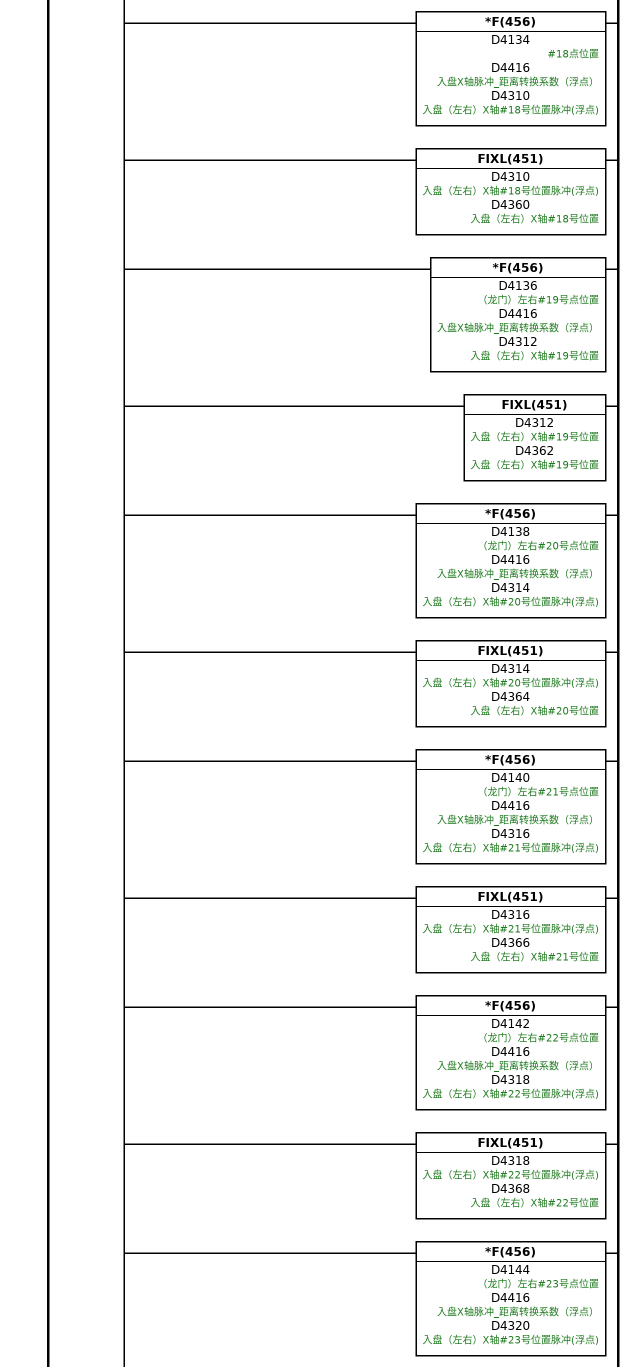

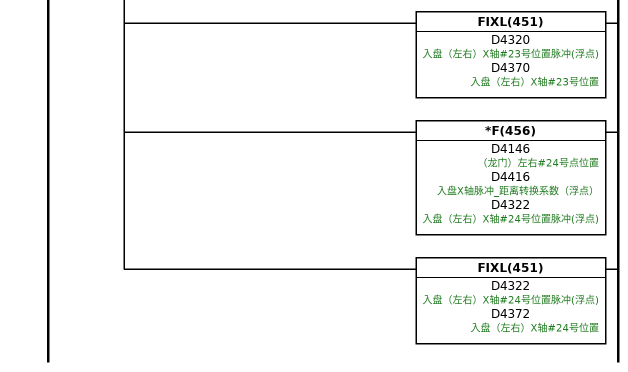
; rung 32: （龙门）左右料机械手各点位置脉冲 / 2排12点
LD P_On
*F(456) D4124 D4416 D4300  ; （龙门）左右#13号点位置, 入盘X轴脉冲_距离转换系数（浮点）, 入盘（左右）X轴#13号位置脉冲(浮点)
FIXL(451) D4300 D4350  ; 入盘（左右）X轴#13号位置脉冲(浮点), 入盘（左右）X轴#13号位置脉冲
*F(456) D4126 D4416 D4302  ; #14号点位置, 入盘X轴脉冲_距离转换系数（浮点）, 入盘（左右）X轴#14号位置脉冲(浮点)
FIXL(451) D4302 D4352  ; 入盘（左右）X轴#14号位置脉冲(浮点), 入盘（左右）X轴#14号位置脉冲
*F(456) D4128 D4416 D4304  ; （龙门）左右#15号点位置, 入盘X轴脉冲_距离转换系数（浮点）, 入盘（左右）X轴#15号位置脉冲(浮点)
FIXL(451) D4304 D4354  ; 入盘（左右）X轴#15号位置脉冲(浮点), 入盘（左右）X轴#15号位置
*F(456) D4130 D4416 D4306  ; （龙门）左右#16号点位置, 入盘X轴脉冲_距离转换系数（浮点）, 入盘（左右）X轴#16号位置脉冲(浮点)
FIXL(451) D4306 D4356  ; 入盘（左右）X轴#16号位置脉冲(浮点), 入盘（左右）X轴#16号位置
*F(456) D4132 D4416 D4308  ; （龙门）左右#17号点位置, 入盘X轴脉冲_距离转换系数（浮点）, 入盘（左右）X轴#17号位置脉冲(浮点)
FIXL(451) D4308 D4358  ; 入盘（左右）X轴#17号位置脉冲(浮点), 入盘（左右）X轴#17号位置脉冲
*F(456) D4134 D4416 D4310  ; #18点位置, 入盘X轴脉冲_距离转换系数（浮点）, 入盘（左右）X轴#18号位置脉冲(浮点)
FIXL(451) D4310 D4360  ; 入盘（左右）X轴#18号位置脉冲(浮点), 入盘（左右）X轴#18号位置
*F(456) D4136 D4416 D4312  ; （龙门）左右#19号点位置, 入盘X轴脉冲_距离转换系数（浮点）, 入盘（左右）X轴#19号位置
FIXL(451) D4312 D4362  ; 入盘（左右）X轴#19号位置
*F(456) D4138 D4416 D4314  ; （龙门）左右#20号点位置, 入盘X轴脉冲_距离转换系数（浮点）, 入盘（左右）X轴#20号位置脉冲(浮点)
FIXL(451) D4314 D4364  ; 入盘（左右）X轴#20号位置脉冲(浮点), 入盘（左右）X轴#20号位置
*F(456) D4140 D4416 D4316  ; （龙门）左右#21号点位置, 入盘X轴脉冲_距离转换系数（浮点）, 入盘（左右）X轴#21号位置脉冲(浮点)
FIXL(451) D4316 D4366  ; 入盘（左右）X轴#21号位置脉冲(浮点), 入盘（左右）X轴#21号位置
*F(456) D4142 D4416 D4318  ; （龙门）左右#22号点位置, 入盘X轴脉冲_距离转换系数（浮点）, 入盘（左右）X轴#22号位置脉冲(浮点)
FIXL(451) D4318 D4368  ; 入盘（左右）X轴#22号位置脉冲(浮点), 入盘（左右）X轴#22号位置
*F(456) D4144 D4416 D4320  ; （龙门）左右#23号点位置, 入盘X轴脉冲_距离转换系数（浮点）, 入盘（左右）X轴#23号位置脉冲(浮点)
FIXL(451) D4320 D4370  ; 入盘（左右）X轴#23号位置脉冲(浮点), 入盘（左右）X轴#23号位置
*F(456) D4146 D4416 D4322  ; （龙门）左右#24号点位置, 入盘X轴脉冲_距离转换系数（浮点）, 入盘（左右）X轴#24号位置脉冲(浮点)
FIXL(451) D4322 D4372  ; 入盘（左右）X轴#24号位置脉冲(浮点), 入盘（左右）X轴#24号位置

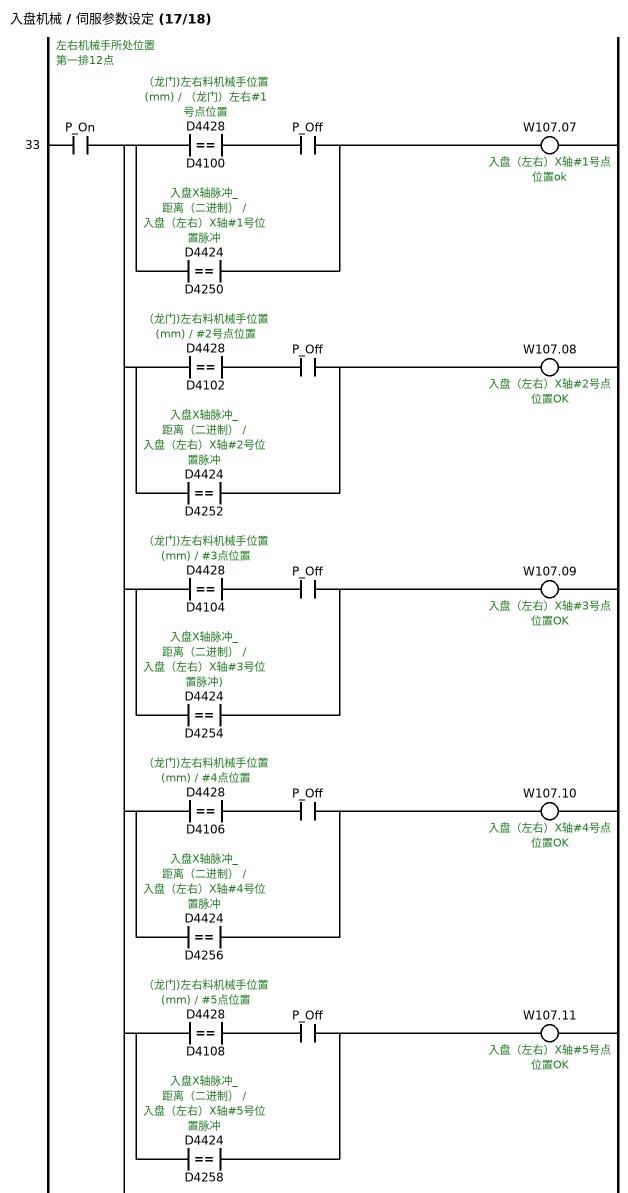

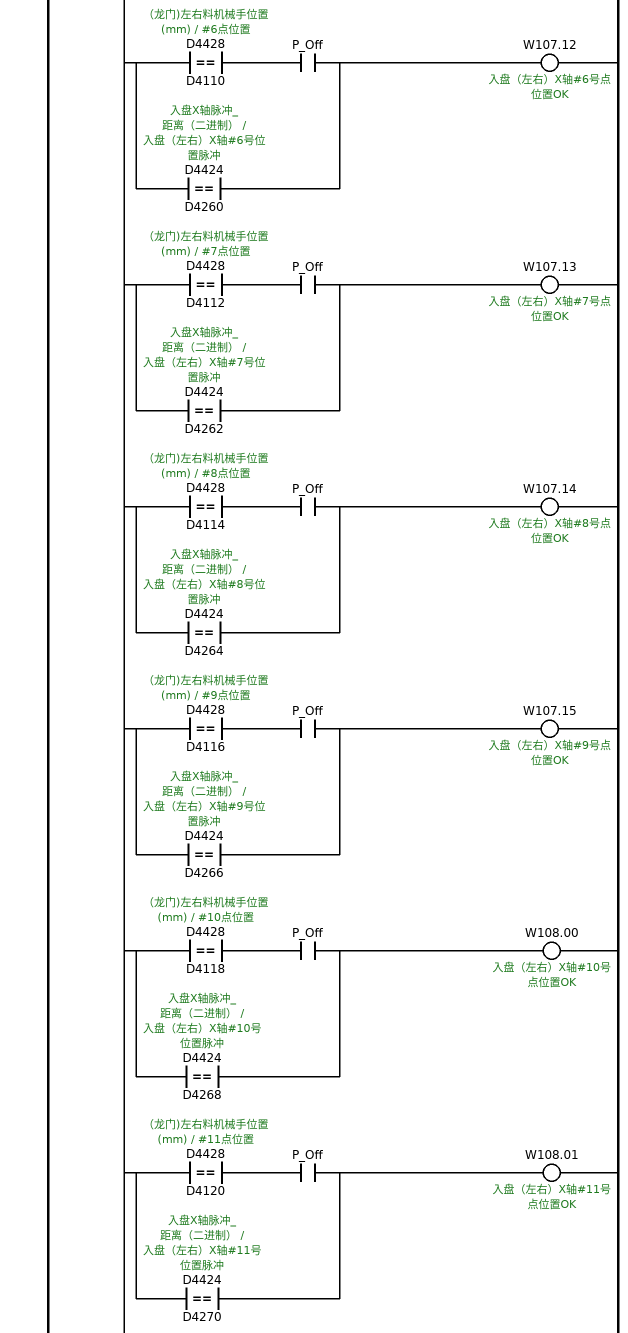

